// TwinCAT 3 PLC project StateMachines
// ProgramVersion: 3.1.4024.0
// libraries:
//   Tc2_Standard, * (Beckhoff Automation GmbH)
//   Tc2_System, * (Beckhoff Automation GmbH)
//   Tc3_Module, * (Beckhoff Automation GmbH)
//   VisuDialogs, * (System)
// project tree:
//   / GlobalTextList.TcGTLO, PlcTask.TcTTO, Visualization Manager.TcVMO (not stored)
//   POUs/ Blinker.TcPOU, MAIN.TcPOU, TrafficLight.TcPOU, TrafficLight2nd.TcPOU, TrafficLightFB.TcPOU, Visualization.TcVIS

CONFIGURATION StateMachines
    RESOURCE PLC ON TwinCAT3
        TASK PlcTask(INTERVAL := T#10ms, PRIORITY := 20);
        PROGRAM MAIN WITH PlcTask : MAIN;
    END_RESOURCE
END_CONFIGURATION

// ---- POUs/MAIN.TcPOU
PROGRAM MAIN
VAR
END_VAR

TrafficLight();

END_PROGRAM

// ---- POUs/TrafficLight.TcPOU
PROGRAM TrafficLight
VAR
	fbTraffic1 : TrafficLightFB; //declaring the function block in the program
	fbTraffic2 : TrafficLight2nd; //declaring the 2nd traffic light
	
	iRedColor : INT;  //integers connected with the hmi that control how much time we input (1st traffic light)
	iYellowColor : INT;
	iGreenColor : INT; 
	
	bRedLight AT %Q* : BOOL; //bool variables that turn the lights on/off through the hmi
	bYellowLight AT %Q* : BOOL;
	bGreenLight AT %Q* : BOOL;
	
	bRedLight2nd AT %Q* : BOOL; //bool variables for the lights of the 2nd traffic light
	bYellowLight2nd : BOOL;
	bGreenLight2nd : BOOL;
	
	bTurnOn AT %I* : BOOL; //bool variable that turns the traffic light on/off
	bTurnOnVis : BOOL; //turns on the visualization
	
	bTextError : BOOL; //bool variable that makes the textbox for error visible/invisible
END_VAR

//1st traffic light
fbTraffic1.iRedIn := iRedColor; //inputing the integers from the hmi to the function
fbTraffic1.iYellowIn := iYellowColor;
fbTraffic1.iGreenIn := iGreenColor;

fbTraffic1.bHardwareON := bTurnOn;
fbTraffic1.bStart := bTurnOnVis; //inputing the status of the traffic light (on/off)

bTextError := fbTraffic1.bError; //outputing the error bool vaiables

bRedLight := fbTraffic1.bRed; //the bool variables take the status for the lights and switch them on/off accordingly
bYellowLight := fbTraffic1.bYellow;
bGreenLight := fbTraffic1.bGreen;

//2nd traffic light
fbTraffic2.iRedIn := iGreenColor; //inputing the integers from the hmi to the function
fbTraffic2.iYellowIn := iYellowColor;
fbTraffic2.iGreenIn := iRedColor; //we reverse the values for red and green so they are in sync and it doesn't make an error

fbTraffic2.bStart := bTurnOnVis; //inputing the status of the traffic light (on/off)

fbTraffic2.bHardwareON := bTurnOn; //we turn on the 2nd traffic light

bTextError := fbTraffic2.bError; //same error as the 1st one

bRedLight2nd := fbTraffic2.bRed; //the bool variables take the status for the lights and switch them on/off accordingly
bYellowLight2nd := fbTraffic2.bYellow;
bGreenLight2nd := fbTraffic2.bGreen;

fbTraffic1(); // calling the function block
fbTraffic2();

END_PROGRAM

// ---- POUs/TrafficLightFB.TcPOU
FUNCTION_BLOCK TrafficLightFB
VAR_INPUT
	bStart : BOOL; //bool variable thats connected with the traffic light status in the program

	iRedIn : INT; //integer variables connected with the time duration integers in the program
	iYellowIn : INT;
	iGreenIn : INT;
	
	bHardwareON : BOOL; //temporary bool for on/off
END_VAR
VAR_OUTPUT
	bRed : BOOL;  // bool variables which output the state of the lights (on/off)
	bYellow : BOOL;
	bGreen : BOOL;
	
	bError : BOOL;	 //error bool variable if true makes the error visible/ivisible	
END_VAR
VAR
	fbTimerSt : TON; //timers for every light time duration
	fbTimerRed : TON; 
	fbTimerYR : TON; 
	fbTimerGreen : TON;
	fbTimerYellow : TON; 
	
	fbTemp1 : TON; //timers for blinking
	fbTemp4 : TON;
	
	fbBlinker : Blinker;
	
		
	iState : UDINT; //state variable to control the states
	
	tTimeRed : TIME; //time variables for the timers
	tTimeYellow : TIME;
	tTimeGreen : TIME;	
	
	fbHardwareTurnON : R_TRIG;
	fbHardwareTurnOFF : TON;
END_VAR

tTimeGreen := INT_TO_TIME(iGreenIn*1000); //coverting the integer values inputet by the user to time variables
tTimeRed := INT_TO_TIME(iRedIn*1000+3230); 
tTimeYellow := INT_TO_TIME(iYellowIn*1000);		
/////////////////////////////////////////////////////
fbHardwareTurnON(CLK := bHardwareON); //if the button is pressed turn on
IF fbHardwareTurnON.Q THEN
	bStart := TRUE;
END_IF
fbHardwareTurnOFF.IN := bHardwareON; //if you hold it for 3s turn off
IF fbHardwareTurnOFF.Q THEN
	bStart := FALSE;
END_IF
/////////////////////////////////////////////////////
	
CASE iState OF
	0: //first state, checks the basic condition
		IF iRedIn > iYellowIn AND iGreenIn > iYellowIn THEN //if the input for yellow is lower than those for green and red execute
			IF bStart THEN
				fbTimerSt.IN := TRUE;//we start the traffic light (set the starting timer)
				iState := 10; //set the next state
				bError := FALSE;
			ELSE
				bRed := FALSE;
				bYellow := FALSE; //if its not started keep the lights turned off
				bGreen := FALSE;
				bError := FALSE;
			END_IF			
		ELSE
			bError := TRUE; //otherwise show an error message
			bYellow := fbBlinker.bBlink; //if there is an error make the yellow light blink
			fbBlinker();
		END_IF
	
	10: //red light
		IF fbTimerSt.Q THEN //if the starting timer elapsed continue
			bRed := TRUE; 
			fbTimerRed.IN := TRUE;	 //we light the red and set the timer to true, also we reset the previous timer
			fbTimerSt.IN := FALSE;
			iState := 20; // go to the next state
		END_IF
	20: //yellow and red light
		IF fbTimerRed.Q THEN
			bYellow := TRUE;
			fbTimerYR.IN := TRUE;
			fbTimerRed.IN := FALSE; //we light the yellow as well, start the yellow/red timer and reset the red timer
			iState := 30; //go to the next state
		END_IF
	30:// green light
		IF fbTimerYR.Q THEN
			bYellow := FALSE;
			bRed := FALSE;
			bGreen := TRUE;
			fbTimerGreen.IN := TRUE; //we turn the red and yellow off and light the green, also we start the green timer but reset the yellow one
			fbTimerYR.IN := FALSE;
			iState := 40; //go to the next state
		END_IF	
	40:// blinker
		IF fbTimerGreen.Q THEN
			bGreen := FALSE;
			fbTemp1.IN := TRUE;
			fbTimerGreen.IN := FALSE; //we turn the green light off for a split second
			iState := 50; //next state
		END_IF
	50: //blinker
		IF fbTemp1.Q THEN
			fbTemp4.IN := TRUE;
			bGreen := fbBlinker.bBlink; //start the blinker on the green light
			fbBlinker();
			IF fbTemp4.Q THEN
				iState := 60; //when the blinker is finished go to the next state
			END_IF	
		END_IF
	60: //yellow light
			bGreen := FALSE; 
			bYellow := TRUE; //we turn the green light off and turn the yellow one on
			fbTimerYellow.IN := TRUE; //we start the yellow timer and reset the last blinking timer
			fbTemp4.IN := FALSE;
			iState := 70; //next state	
	70: //reset the yellow timer and go back to state 0
		IF fbTimerYellow.Q THEN
			bYellow := FALSE;
			fbTimerYellow.IN := FALSE;
			iState := 0;	
		END_IF
END_CASE

fbHardwareTurnOFF(PT := T#3000MS);

fbTemp4(PT := T#3200MS);

fbTemp1(PT := T#30MS);
fbTimerSt(PT := T#50MS); //timer for start
fbTimerRed(PT := tTimeRed); //timer for red
fbTimerYR(PT := tTimeYellow); //timer for yellow
fbTimerGreen(PT := tTimeGreen); //timer for green
fbTimerYellow(PT := tTimeYellow); //timer for yellow 2nd cicle

END_FUNCTION_BLOCK

// ---- POUs/Blinker.TcPOU
FUNCTION_BLOCK Blinker
VAR_INPUT
END_VAR
VAR_OUTPUT
	bBlink : BOOL; //bool variable that sets the light on/off constantly
END_VAR
VAR
	fbTimer1 : TON;
	fbTimer2 : TON;
	fbTimer3 : TON;
	
	iStateFB : INT; //state variable to switch between states in the blinker function block
END_VAR

CASE iStateFB OF
	0:
		bBlink := TRUE;
		fbTimer1.IN := TRUE;
		iStateFB := 10;
	10:	
		IF fbTimer1.Q THEN
			bBlink := FALSE;
			fbTimer1.IN := FALSE;
			fbTimer2.IN := TRUE;
			iStateFB := 20;
		END_IF
	20:
		IF fbTimer2.Q THEN
			bBlink := TRUE;
			fbTimer2.IN := FALSE;
			fbTimer3.IN := TRUE;
			iStateFB := 30;
		END_IF	
	30:
		IF fbTimer3.Q THEN
			bBlink := FALSE;
			fbTimer3.IN := FALSE;
			iStateFB := 0;
		END_IF	
END_CASE

fbTimer1(PT := T#400MS);// timers for blinkers
fbTimer2(PT := T#400MS);
fbTimer3(PT := T#400MS);

END_FUNCTION_BLOCK

// ---- POUs/TrafficLight2nd.TcPOU
FUNCTION_BLOCK TrafficLight2nd
VAR_INPUT
	bStart : BOOL; //bool variable thats connected with the traffic light status in the program

	iRedIn : INT; //integer variables connected with the time duration integers in the program
	iYellowIn : INT;
	iGreenIn : INT;
	
	bHardwareON : BOOL; //temporary bool for on/off
END_VAR
VAR_OUTPUT
	bRed : BOOL;  // bool variables which output the state of the lights (on/off)
	bYellow : BOOL;
	bGreen : BOOL;
	
	bError : BOOL;	 //error bool variable if true makes the error visible/ivisible	
END_VAR
VAR
	fbTimerSt : TON; //timers for every light time duration
	fbTimerRed : TON; 
	fbTimerYR : TON; 
	fbTimerGreen : TON;
	fbTimerYellow : TON; 
	
	fbTemp1 : TON; //timers for blinking
	fbTemp4 : TON;
	
	fbBlinker : Blinker;
	
		
	iState : UDINT; //state variable to control the states
	
	tTimeRed : TIME; //time variables for the timers
	tTimeYellow : TIME;
	tTimeGreen : TIME;	
	
	fbHardwareTurnON : R_TRIG;
	fbHardwareTurnOFF : TON;
END_VAR

tTimeGreen := INT_TO_TIME(iGreenIn*1000); //coverting the integer values inputet by the user to time variables
tTimeRed := INT_TO_TIME(iRedIn*1000+3230); 
tTimeYellow := INT_TO_TIME(iYellowIn*1000);		
/////////////////////////////////////////////////////
fbHardwareTurnON(CLK := bHardwareON); //if the button is pressed turn on
IF fbHardwareTurnON.Q THEN
	bStart := TRUE;
END_IF
fbHardwareTurnOFF.IN := bHardwareON; //if you hold it for 3s turn off
IF fbHardwareTurnOFF.Q THEN
	bStart := FALSE;
END_IF
/////////////////////////////////////////////////////
	
CASE iState OF
	0: //first state, checks the basic condition
		IF iRedIn > iYellowIn AND iGreenIn > iYellowIn THEN //if the input for yellow is lower than those for green and red execute
			IF bStart THEN
				fbTimerSt.IN := TRUE;//we start the traffic light (set the starting timer)
				iState := 10; //set the next state
				bError := FALSE;
			ELSE
				bRed := FALSE;
				bYellow := FALSE; //if its not started keep the lights turned off
				bGreen := FALSE;
				bError := FALSE;
			END_IF			
		ELSE
			bError := TRUE; //otherwise show an error message
			bYellow := fbBlinker.bBlink; //if there is an error make the yellow light blink
			fbBlinker();
		END_IF
	
	10: //green light
		IF fbTimerSt.Q THEN //if the starting timer elapsed continue
			fbTimerYR.IN := FALSE;
			bRed := FALSE;
			bYellow := FALSE;
			bGreen := TRUE; 
			fbTimerGreen.IN := TRUE;	 //reversed the times so it works in sync
			fbTimerSt.IN := FALSE;
			fbTimerRed.IN := FALSE;
			iState := 20; // go to the next state
		END_IF
	20: //blinker
		IF fbTimerGreen.Q THEN
			bGreen := FALSE;
			fbTemp1.IN := TRUE;
			fbTimerGreen.IN := FALSE; //we turn the green light off for a split second
			iState := 30; //next state
		END_IF
	30:
		IF fbTemp1.Q THEN
			fbTemp4.IN := TRUE;
			bGreen := fbBlinker.bBlink; //start the blinker on the green light
			fbBlinker();
			IF fbTemp4.Q THEN
				iState := 40; //when the blinker is finished go to the next state
			END_IF	
		END_IF
	40:
		bGreen := FALSE; 
		bYellow := TRUE; //we turn the green light off and turn the yellow one on
		fbTimerYellow.IN := TRUE; //we start the yellow timer and reset the last blinking timer
		fbTemp4.IN := FALSE;
		iState := 50; //next state
	50:
		IF fbTimerYellow.Q THEN
			bYellow := FALSE;
			fbTimerYellow.IN := FALSE;
			bRed := TRUE;
			fbTimerRed.IN := TRUE;
			iState := 60;
		END_IF
	60:
		IF fbTimerRed.Q THEN
			bYellow := TRUE;
			fbTimerYR.IN := TRUE;
			IF fbTimerYR.Q THEN
				iState := 0;
			END_IF
		END_IF
		
END_CASE

fbHardwareTurnOFF(PT := T#3000MS);

fbTemp4(PT := T#3200MS);

fbTemp1(PT := T#30MS);
fbTimerSt(PT := T#50MS); //timer for start
fbTimerRed(PT := tTimeRed); //timer for red
fbTimerYR(PT := tTimeYellow); //timer for yellow
fbTimerGreen(PT := tTimeGreen); //timer for green
fbTimerYellow(PT := tTimeYellow); //timer for yellow 2nd cicle

END_FUNCTION_BLOCK

// ---- GlobalTextList.TcGTLO
TEXTLIST GlobalTextList
  391 = '%i Green'
  423 = '%i Red'
  73 = '%i Yellow'
  231 = 'CRITICAL ERROR!!!!!'
  858 = 'ERROR!!!!!'
END_TEXTLIST

// ---- POUs/Visualization.TcVIS
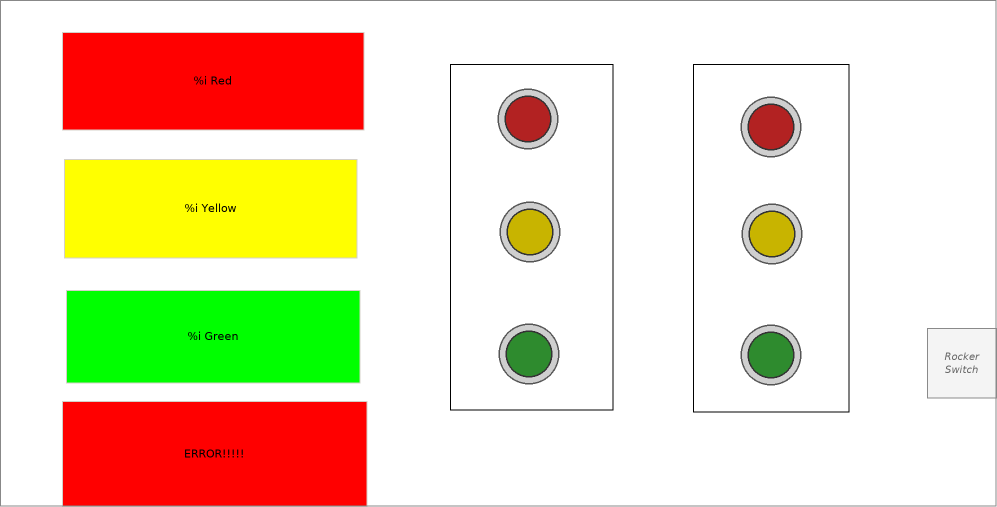
VISUALIZATION Visualization  // 997x507
    Rectangle (450,64 163x346)
    Lamp1 (494,319 70x70), variable: TrafficLight.bGreenLight, style: Lamp-Lamp1-Green
    Lamp1 (495,197 70x70), variable: TrafficLight.bYellowLight, style: Lamp-Lamp1-Yellow
    Lamp1 (493,84 70x70), variable: TrafficLight.bRedLight, style: Lamp-Lamp1-Red
    RockerSwitch (927,328 70x70), variable: TrafficLight.bTurnOnVis, behaviour: TOGGLE, style: Switch-RockerSwitch-Red
    Textfield (62,32 302x98), "%i Red", text variable: TrafficLight.iRedColor
        OnMouseDown: write the text variable via Default
    Textfield (64,159 293x99), "%i Yellow", text variable: TrafficLight.iYellowColor
        OnMouseDown: write the text variable via Default
    Textfield (62,401 305x106), "ERROR!!!!!", invisible if: NOT TrafficLight.bTextError
    Textfield (66,290 294x93), "%i Green", text variable: TrafficLight.iGreenColor
        OnMouseDown: write the text variable via Default
    Rectangle (693,64 156x348)
    Lamp1 (736,92 70x70), variable: TrafficLight.bRedLight2nd, style: Lamp-Lamp1-Red
    Lamp1 (737,199 70x70), variable: TrafficLight.bYellowLight2nd, style: Lamp-Lamp1-Yellow
    Lamp1 (736,320 70x70), variable: TrafficLight.bGreenLight2nd, style: Lamp-Lamp1-Green
END_VISUALIZATION
